FUNCTION_BLOCK FB_GCModuleConfigurationAdapter IMPLEMENTS I_ModuleConfigurationAdapter
VAR
	_SpinAxisBound : ARRAY[1..Param_Config.MaxConfiguredModules] OF BOOL;
	_LiftPinAxisBound : ARRAY[1..Param_Config.MaxConfiguredModules] OF BOOL;
END_VAR

METHOD PUBLIC M_ApplyRuntimeConfig : BOOL
VAR_INPUT
	Slot : UINT;
END_VAR
VAR_IN_OUT CONSTANT
	RuntimeConfig : ST_ModuleRuntimeConfig;
END_VAR
VAR_OUTPUT
	ErrorMessage : STRING(255);
END_VAR
M_ApplyRuntimeConfig := FALSE;
ErrorMessage := '';
IF NOT M_IsSlotSupported(Slot := Slot) THEN
	ErrorMessage := 'GC slot is outside the supported range.';
	RETURN;
END_IF
IF RuntimeConfig.ModuleType <> TO_STRING(E_ModuleType.GC) THEN
	ErrorMessage := 'Runtime configuration type is incompatible with the GC adapter.';
	RETURN;
END_IF
GVL_Module.GC_Runtime[Slot] := RuntimeConfig;
M_ApplyRuntimeConfig := TRUE;
END_METHOD

METHOD PUBLIC M_BindReference : BOOL
VAR_INPUT
	Slot : UINT;
	TargetPort : STRING(80);
	BaseUnit : I_BaseUnit;
END_VAR
VAR_OUTPUT
	ErrorMessage : STRING(255);
END_VAR
VAR
	Port : E_GCReferencePort;
	Axis : I_Axis_BaseUnit;
END_VAR
M_BindReference := FALSE;
ErrorMessage := '';
IF NOT M_IsSlotSupported(Slot := Slot) THEN
	ErrorMessage := 'GC slot is outside the supported range.';
	RETURN;
END_IF
IF BaseUnit = 0 THEN
	ErrorMessage := 'Cannot bind an unbound BaseUnit reference.';
	RETURN;
END_IF

Port := E_GCReferencePort.Unknown;
IF TargetPort = TO_STRING(E_GCReferencePort.SpinAxis_BaseUnit) THEN
	Port := E_GCReferencePort.SpinAxis_BaseUnit;
ELSIF TargetPort = TO_STRING(E_GCReferencePort.LiftPinAxis_BaseUnit) THEN
	Port := E_GCReferencePort.LiftPinAxis_BaseUnit;
ELSE
	ErrorMessage := 'Unknown GC reference port.';
	RETURN;
END_IF

Axis := 0;
IF NOT __QUERYINTERFACE(BaseUnit, Axis) THEN
	ErrorMessage := CONCAT('Reference type is incompatible with GC port ', TO_STRING(Port));
	RETURN;
END_IF

CASE Port OF
	E_GCReferencePort.SpinAxis_BaseUnit:
		IF _SpinAxisBound[Slot] THEN
			ErrorMessage := CONCAT('Duplicate GC reference binding for ', TO_STRING(Port));
			RETURN;
		END_IF
		GVL_Module.GC_SpinAxis[Slot] := Axis;
		_SpinAxisBound[Slot] := TRUE;

	E_GCReferencePort.LiftPinAxis_BaseUnit:
		IF _LiftPinAxisBound[Slot] THEN
			ErrorMessage := CONCAT('Duplicate GC reference binding for ', TO_STRING(Port));
			RETURN;
		END_IF
		GVL_Module.GC_LiftPinAxis[Slot] := Axis;
		_LiftPinAxisBound[Slot] := TRUE;
END_CASE
M_BindReference := TRUE;
END_METHOD

METHOD PUBLIC M_ClearSlot : BOOL
VAR_INPUT
	Slot : UINT;
END_VAR
VAR_OUTPUT
	ErrorMessage : STRING(255);
END_VAR
M_ClearSlot := FALSE;
ErrorMessage := '';
IF NOT M_IsSlotSupported(Slot := Slot) THEN
	ErrorMessage := 'GC slot is outside the supported range.';
	RETURN;
END_IF
GVL_Module.GC_SpinAxis[Slot] := 0;
GVL_Module.GC_LiftPinAxis[Slot] := 0;
MEMSET(ADR(GVL_Module.GC_Runtime[Slot]), 0, SIZEOF(GVL_Module.GC_Runtime[Slot]));
_SpinAxisBound[Slot] := FALSE;
_LiftPinAxisBound[Slot] := FALSE;
M_ClearSlot := TRUE;
END_METHOD

METHOD PUBLIC M_IsSlotSupported : BOOL
VAR_INPUT
	Slot : UINT;
END_VAR
M_IsSlotSupported := (Slot >= 1) AND (Slot <= Param_Config.MaxConfiguredModules);
END_METHOD

METHOD PUBLIC M_RegisterIo : BOOL
VAR_INPUT
	Slot : UINT;
END_VAR
VAR_IN_OUT
	LinkVariableManager : FB_LinkVariableManager;
END_VAR
VAR_OUTPUT
	ModuleSymbol : STRING(255);
	ErrorMessage : STRING(255);
END_VAR
M_RegisterIo := FALSE;
ModuleSymbol := '';
ErrorMessage := '';
IF NOT M_IsSlotSupported(Slot := Slot) THEN
	ErrorMessage := 'GC slot is outside the supported range.';
	RETURN;
END_IF
IF NOT LinkVariableManager.M_RegisterGCModule(
	Module := GVL_Module.GC[Slot],
	ModuleSymbol => ModuleSymbol) THEN
	ErrorMessage := LinkVariableManager.ErrorMessage;
	RETURN;
END_IF
M_RegisterIo := TRUE;
END_METHOD

METHOD PUBLIC M_ValidateReferences : BOOL
VAR_INPUT
	Slot : UINT;
END_VAR
VAR_OUTPUT
	ErrorMessage : STRING(255);
END_VAR
M_ValidateReferences := FALSE;
ErrorMessage := '';
IF NOT M_IsSlotSupported(Slot := Slot) THEN
	ErrorMessage := 'GC slot is outside the supported range.';
	RETURN;
END_IF
IF NOT _SpinAxisBound[Slot] THEN
	ErrorMessage := CONCAT('Missing required GC reference port ', TO_STRING(E_GCReferencePort.SpinAxis_BaseUnit));
	RETURN;
END_IF
IF NOT _LiftPinAxisBound[Slot] THEN
	ErrorMessage := CONCAT('Missing required GC reference port ', TO_STRING(E_GCReferencePort.LiftPinAxis_BaseUnit));
	RETURN;
END_IF
M_ValidateReferences := TRUE;
END_METHOD

END_FUNCTION_BLOCK

(* stored: Version 1.1.0.1, ProductVersion 3.1.4026.18
   POU FB_GCModuleConfigurationAdapter: Id {d1ed4bb2-81ea-4b79-900f-c662788b8aa5}, SpecialFunc None
   Method M_ApplyRuntimeConfig: Id {3fe7b39d-d396-4fb1-a765-1f717436db5b}
   Method M_BindReference: Id {415cb1e9-35c4-4435-8776-527c38751fd5}
   Method M_ClearSlot: Id {3eff8948-41a3-47d4-b197-f93e2ec9fbf1}
   Method M_IsSlotSupported: Id {59dbc889-0ba5-462f-b874-f60410801f22}
   Method M_RegisterIo: Id {afcdad32-5005-4810-bb84-67a02f90ef60}
   Method M_ValidateReferences: Id {3598c4ac-0cd5-4fc2-b868-fb2f7dc5dac3} *)
